// TIA Portal V16 program export: 1 tag tables, 0 data types, 3 data blocks, 4 code blocks (in call order from the OBs), 0 instance data blocks

VAR_GLOBAL   // PLC tag table "Default tag table"
   estop_clear AT %I0.0 : Bool;   //    {ExternalAccessible false, ExternalVisible false, ExternalWritable false}
   interlock AT %Q0.0 : Bool;   //    {ExternalAccessible false, ExternalVisible false, ExternalWritable false}
   reset AT %I0.1 : Bool;   //    {ExternalAccessible false, ExternalVisible false, ExternalWritable false}
END_VAR

DATA_BLOCK "DataFromSafety"
{ S7_Optimized_Access := 'TRUE' }
VERSION : 0.1
NON_RETAIN
   VAR 
      running : Bool;
   END_VAR


BEGIN

END_DATA_BLOCK

DATA_BLOCK "DataToSafety"
{ S7_Optimized_Access := 'TRUE' }
VERSION : 0.1
NON_RETAIN
   VAR 
      run : Bool;
   END_VAR


BEGIN

END_DATA_BLOCK

DATA_BLOCK "Main_Safety_RTG1_DB"
{ S7_Optimized_Access := 'TRUE' }
NAME : FUSI
VERSION : 0.1
NON_RETAIN
"Main_Safety_RTG1"

BEGIN

END_DATA_BLOCK

ORGANIZATION_BLOCK "Main"   // OB1, LAD, ProgramCycle
TITLE = "Main Program Sweep (Cycle)"
{ S7_Optimized_Access := 'TRUE' }
VERSION : 0.1
// stored: AutoNumber true, IsIECCheckEnabled false, SetENOAutomatically false
   VAR_INPUT
      Initial_Call : Bool;   // Initial call of this OB
      Remanence : Bool;   // =True, if remanent data are available
   END_VAR
BEGIN
END_ORGANIZATION_BLOCK

FUNCTION_BLOCK "Main_Safety_RTG1"   // FB1, F_FBD
{ S7_Optimized_Access := 'TRUE' }
VERSION : 0.1
// stored: AutoNumber false, IsIECCheckEnabled false, UDAEnableTagReadback false
   VAR
      faults_clear : Bool;
      last_estop_clear : Bool;
      last_reset : Bool;
   END_VAR
   VAR_TEMP   // added for the SCL form of the ladder/FBD networks
      _w1 : Bool;
      _w2 : Bool;
   END_VAR
BEGIN

REGION Network 1
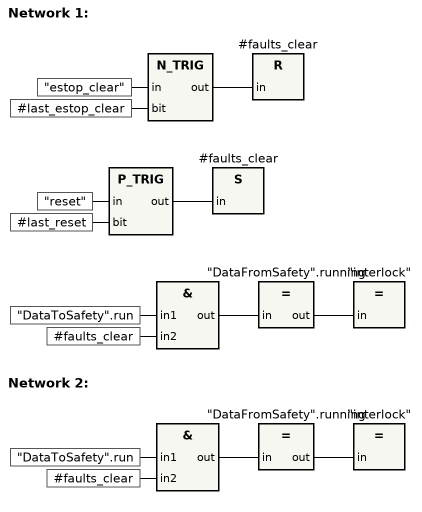
   #_w1 := NOT "estop_clear" AND #last_estop_clear;   // falling edge
   #last_estop_clear := "estop_clear";
   IF #_w1 THEN #faults_clear := FALSE; END_IF;
   #_w2 := "reset" AND NOT #last_reset;   // rising edge
   #last_reset := "reset";
   IF #_w2 THEN #faults_clear := TRUE; END_IF;
   "DataFromSafety".running := "DataToSafety".run AND #faults_clear;
   "interlock" := "DataFromSafety".running;
END_REGION

REGION Network 2
   "DataFromSafety".running := "DataToSafety".run AND #faults_clear;
   "interlock" := "DataFromSafety".running;
END_REGION
END_FUNCTION_BLOCK

FUNCTION_BLOCK "Step1"   // FB3, F_FBD
{ S7_Optimized_Access := 'TRUE' }
VERSION : 0.1
// stored: AutoNumber true, IsIECCheckEnabled false, UDAEnableTagReadback false
BEGIN

REGION Network 1
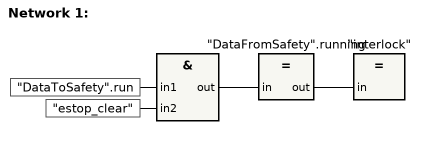
   "DataFromSafety".running := "DataToSafety".run AND "estop_clear";
   "interlock" := "DataFromSafety".running;
END_REGION
END_FUNCTION_BLOCK

FUNCTION_BLOCK "Step2"   // FB2, F_FBD
{ S7_Optimized_Access := 'TRUE' }
VERSION : 0.1
// stored: AutoNumber true, IsIECCheckEnabled false, UDAEnableTagReadback false
   VAR
      faults_clear : Bool;
      last_estop_clear : Bool;
      last_reset : Bool;
   END_VAR
   VAR_TEMP   // added for the SCL form of the ladder/FBD networks
      _w1 : Bool;
      _w2 : Bool;
   END_VAR
BEGIN

REGION Network 1
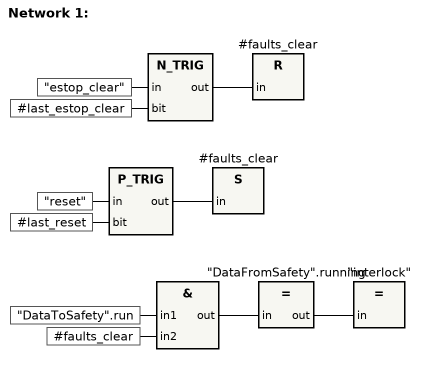
   #_w1 := NOT "estop_clear" AND #last_estop_clear;   // falling edge
   #last_estop_clear := "estop_clear";
   IF #_w1 THEN #faults_clear := FALSE; END_IF;
   #_w2 := "reset" AND NOT #last_reset;   // rising edge
   #last_reset := "reset";
   IF #_w2 THEN #faults_clear := TRUE; END_IF;
   "DataFromSafety".running := "DataToSafety".run AND #faults_clear;
   "interlock" := "DataFromSafety".running;
END_REGION
END_FUNCTION_BLOCK
